// TIA Portal V20 export
DATA_BLOCK "Config"   // DB135
// stored: Access Published, MemoryReserve 100, Namespace Unit1.Em13
   VAR
      em : "LAF_typeEmConfiguration";   // Configuration of EM Parameters
      axis : Array[0.._.U1EM13_NO_OF_AXES] of DB_ANY;
      cmJRUnloadingPnPSafetyPin : "LBC_typeDigitalSignalConfiguration";
      cmJRUnloadingPnPJRDetect : "LBC_typeDigitalSignalConfiguration";
   END_VAR
   VAR RETAIN
      cmJRUnloadingPnPAxisX : "LBC_typeAxis64PosConfiguration";
      cmJRUnloadingPnPAxisZ : "LBC_typeAxis64PosConfiguration";
      cmJRUnloadingPnPAxisC : "LBC_typeAxis64PosConfiguration";
   END_VAR
   VAR
      cmJRUnloadingPnPClampOpenClose : "LBC_typeTwoWayActuatorConfiguration";
      softcam : Struct
         JRUnloadingPnPAxisX : "LER_typeSoftCamInterface";
         JRUnloadingPnPAxisZ : "LER_typeSoftCamInterface";
         JRUnloadingPnPAxisC : "LER_typeSoftCamInterface";
      END_STRUCT;
   END_VAR
BEGIN
   em.referenceDesignator.parent := WSTRING#'U1';
   em.referenceDesignator.relative := WSTRING#'EM0';
   cmJRUnloadingPnPAxisX.referenceDesignator := WSTRING#'UNLOADING P&P X-Axis';
   cmJRUnloadingPnPAxisZ.referenceDesignator := WSTRING#'UNLOADING P&P Z-Axis';
   cmJRUnloadingPnPAxisC.referenceDesignator := WSTRING#'UNLOADING P&P C-Axis';
   cmJRUnloadingPnPClampOpenClose.referenceDesignator := WSTRING#'UNLOADING P&P CLAMP';
   cmJRUnloadingPnPClampOpenClose.monitoringDiscrepancy := T#5s;
END_DATA_BLOCK
